# EPICS StreamDevice protocol: knrk6Sup/knrk6.proto
Terminator = CR;
ReplyTimeout = 10000;
LockTimeout = 20000;

get_position {
    out "p";
    in "%i";
}

set_position {
    out "%i";
    in "OK";
}

get_valve {
    out "t";
    in "VALVE %i";
}

readError {
    in "E%d";
}
